PROGRAM MAIN
VAR
	fbPayload_1 : Payload;
	fbPayload_2 : Payload;
	bStart,bStart2,bStart3 : BOOL;
	Size1,Size2,Size3,Size4 : UINT;
	
	pBuffer : POINTER TO BYTE;
	aMarshalBuffer : ARRAY[0..1999] OF BYTE;
	
END_VAR

fbPayload_1();
fbPayload_2();
IF 	bStart
	THEN
	
	
	pBuffer := fbPayload_2.Desirialize(fbPayload_1.Serialize());
	__DELETE(pBuffer);
	bStart := FALSE;
	
END_IF

IF	bStart2
	THEN
	
	
	pBuffer := fbPayload_1.Serialize();
	MEMCPY(ADR(aMarshalBuffer),pBuffer,fbPayload_1.nObjectSize);
	__DELETE(pBuffer);
	bStart2 := FALSE;
END_IF

IF	bStart3
	THEN
	fbPayload_2.Desirialize(ADR(aMarshalBuffer));
	//MEMCPY(ADR(fbPayload_2),ADR(aMarshalBuffer),fbPayload_2.nObjectSize);
	bStart3 := FALSE;
END_IF

END_PROGRAM

(* stored: Version 1.1.0.1, ProductVersion 3.1.4024.2
   POU MAIN: Id {a428ac16-d16d-414b-aa2c-821dfdc90fce}, SpecialFunc None *)
